FUNCTION_BLOCK ABSTRACT StateMachine
VAR_INPUT
END_VAR
VAR_OUTPUT
	eStateMachine : E_StateMachine;
END_VAR
VAR
	stStateMachine : ST_StateMachine;
END_VAR

CASE eStateMachine OF

	eInit:
		Init();
	eBusy:
		Busy();
	eIdle:
		Idle();
	eReady:
		Ready();
	eWaiting:
		Waiting();
	eError:
		Error();
		
END_CASE

METHOD ABSTRACT Busy : BOOL
VAR_INPUT
END_VAR
END_METHOD

METHOD PRIVATE ChangeState : BOOL
VAR_INPUT
	eStateMachine : E_StateMachine;
END_VAR
THIS^.eStateMachine := eStateMachine;
END_METHOD

METHOD ABSTRACT Error : BOOL
VAR_INPUT
END_VAR
END_METHOD

METHOD ABSTRACT Idle : BOOL
VAR_INPUT
END_VAR
END_METHOD

METHOD ABSTRACT Init : BOOL
VAR_INPUT
END_VAR
END_METHOD

METHOD ABSTRACT Ready : BOOL
VAR_INPUT
END_VAR
END_METHOD

METHOD ABSTRACT Waiting : BOOL
VAR_INPUT
END_VAR
END_METHOD

END_FUNCTION_BLOCK

(* stored: Version 1.1.0.1, ProductVersion 3.1.4024.0
   POU StateMachine: Id {11f3d975-8a9c-42f7-90c3-a017c227a81f}, SpecialFunc None
   Method Busy: Id {b89fd49e-6e72-444b-a1c1-9076acdfc55f}
   Method ChangeState: Id {cacbdf26-de46-4210-84d6-77db883ad517}
   Method Error: Id {a5919321-1ff0-46ee-ae01-6220d4cc812c}
   Method Idle: Id {5173a18e-95d9-4e4c-8494-dd70cd7612c7}
   Method Init: Id {9e74f0af-aa5a-4fcb-aa76-2d2219c451fb}
   Method Ready: Id {1fb937da-5310-497e-877e-071145bd9b89}
   Method Waiting: Id {0f01fbf9-d0ef-4dcc-8adf-961ac51a17ff} *)
